SUBAPPLICATION mapping_aux (* Subapplication Type *)
  (* Standard: 61499-2 *)
  (* Version 1.0, 2023-01-29, Franz *)
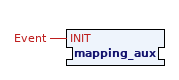
  EVENT_INPUT
    INIT;
  END_EVENT
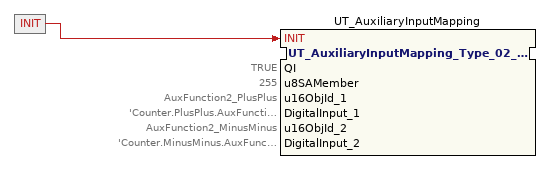
  FBS
    UT_AuxiliaryInputMapping : UT_AuxiliaryInputMapping_Type_02_Bool_NonLatched(QI := TRUE, u8SAMember := 255, u16ObjId_1 := AuxFunction2_PlusPlus, DigitalInput_1 := 'Counter.PlusPlus.AuxFunction2', u16ObjId_2 := AuxFunction2_MinusMinus, DigitalInput_2 := 'Counter.MinusMinus.AuxFunction2');
  END_FBS
  EVENT_CONNECTIONS
    INIT TO UT_AuxiliaryInputMapping.INIT;
  END_CONNECTIONS
END_SUBAPPLICATION
